FUNCTION_BLOCK FB_Observer_DWORD EXTENDS FB_AbstractObserver
VAR
    _nVal:              DWORD;
END_VAR

METHOD FB_init : BOOL
VAR_INPUT
	bInitRetains : BOOL; // if TRUE, the retain variables are initialized (warm start / cold start)
	bInCopyCode : BOOL;  // if TRUE, the instance afterwards gets moved into the copy code (online change)
END_VAR
THIS^._nTypeClass := __SYSTEM.TYPE_CLASS.TYPE_DWORD;
THIS^._pVal := ADR(THIS^._nVal);
THIS^._nSize := SIZEOF(THIS^._nVal);
END_METHOD

PROPERTY nValue32 : DWORD
GET
nValue32 := THIS^._nVal;
END_GET
END_PROPERTY

END_FUNCTION_BLOCK

(* stored: Version 1.1.0.1, ProductVersion 3.1.4024.12
   POU FB_Observer_DWORD: Id {2211ccfd-2397-0a0a-356c-334227435b2b}, SpecialFunc None
   Method FB_init: Id {e58059c5-96ef-000b-3fff-07ab4cf43fc6}
   Property nValue32: Id {283d9a4b-902e-0f81-0a11-0f77da394489}
   Get Get: Id {e0d1ce6c-21e1-0b2d-15f3-6bef417c399e} *)
